PROGRAM AlargEx
VAR
	bInit			: BOOL := TRUE;
	bRaise			: BOOL;
	bClear			: BOOL;
	
	fbAlm			: FB_TcAlarm;
	fbSourceInfo	: FB_TcSourceInfo;
END_VAR

IF bInit THEN
	bInit := FALSE;
	
	fbSourceInfo.Clear();
	fbSourceInfo.sName := '%l%L_MyName%/l%';
	
	//fbAlm.CreateEx(TC_Events.MyEventClass.MyAlarm, TRUE, 0);
	fbAlm.CreateEx(TC_Events.MyEventClass.MyFirstAlarm, TRUE, fbSourceInfo);
	
	fbAlm.ipArguments.Clear();
	fbAlm.ipArguments.AddString('BMK');
END_IF

IF bRaise THEN
	bRaise := FALSE;
	fbAlm.Raise(0);
END_IF

IF bClear AND (fbAlm.eConfirmationState = TcEventConfirmationState.Confirmed) THEN
	bClear := FALSE;
	fbAlm.Clear(0, FALSE);
END_IF

END_PROGRAM

(* stored: Version 1.1.0.1, ProductVersion 3.1.4024.12
   POU AlargEx: Id {806ffe9a-70c8-4db3-b35f-4fbb1bfb96d1}, SpecialFunc None *)
